{attribute 'GeneratedUsingTerminal: EK1122-0000-0018'}
{attribute addProperty BoxType "EK1122-0000-0018"}
{attribute addProperty Id "Beckhoff_EL30xxsub_EK1100EK1100_1FC0878B2"}
{attribute addProperty CRC "1837458359"}
{attribute addProperty Size "2"}
TYPE Beckhoff_EL30xxEK1122_6D8563B7 EXTENDS EK1122_1FC0878B :
STRUCT
	{attribute addProperty Name "Beckhoff_EL30xxsub_EK1100"}
	Beckhoff_EL30xxsub_EK1100 : EK1100_1FC0878B;
END_STRUCT
END_TYPE

(* stored: Version 1.2.0.0, ProductVersion 3.1.4024.9
   DUT Beckhoff_EL30xxEK1122_6D8563B7: Id {ee092e6a-22a6-4ee4-83be-8ae308ca41f2} *)
